Staubli VAL3: onRun.pgx

public program onRun(string& x_sItem[])
  local num l_nCount
  local string l_sItem[3]
  local num l_nFlag
  local bool l_bMode[3]
  local bool l_bActive
  local bool l_bFound
  local num l_nSize
  local num i
  local num j
  local string l_sName
  local string l_sMessage
begin
  //
  // find how many time and fill sItem and l_bMode
  //
  l_nCount=-1
  do
    l_nCount=l_nCount+1
    // sMode
    i=find(x_sItem,"AND")
    if i!=-1
      i=i+len("AND")+1
    endIf
    //
    if i!=-1
      l_sItem[l_nCount]=left(x_sItem,i)
      x_sItem=right(x_sItem,len(x_sItem)-i)
    else
      l_sItem[l_nCount]=x_sItem
    endIf
    l_nFlag=find(l_sItem[l_nCount],">")
    // l_bMode
    if find(l_sItem[l_nCount],">ON")!=-1
      l_bMode[l_nCount]=true
    else
      l_bMode[l_nCount]=false
    endIf
    //sItem
    l_sItem[l_nCount]=left(l_sItem[l_nCount],l_nFlag)
  until i==-1
  //
  // set the OUTPUT wait for the output
  //
  call getSize(l_nSize)
  for i=0 to l_nCount
    // execute
    l_sName=l_sItem[i]
    if saveInOut:dOutput[l_sName].bEnable
      saveInOut:dOutput[l_sName].dDio=l_bMode[i]
    endIf
  endFor
end
